TYPE T_Ctrl_SIf_JUN_In :
STRUCT
	///sensor hanger passed the junction
	bolPassed: Base_PLC.T_Ctrl_IoBoolDebounced;
END_STRUCT
END_TYPE

(* stored: Version 1.1.0.1, ProductVersion 3.1.0.23
   DUT T_Ctrl_SIf_JUN_In: Id {67dd8e32-3efc-4f22-acdb-e6ee6d753643} *)
